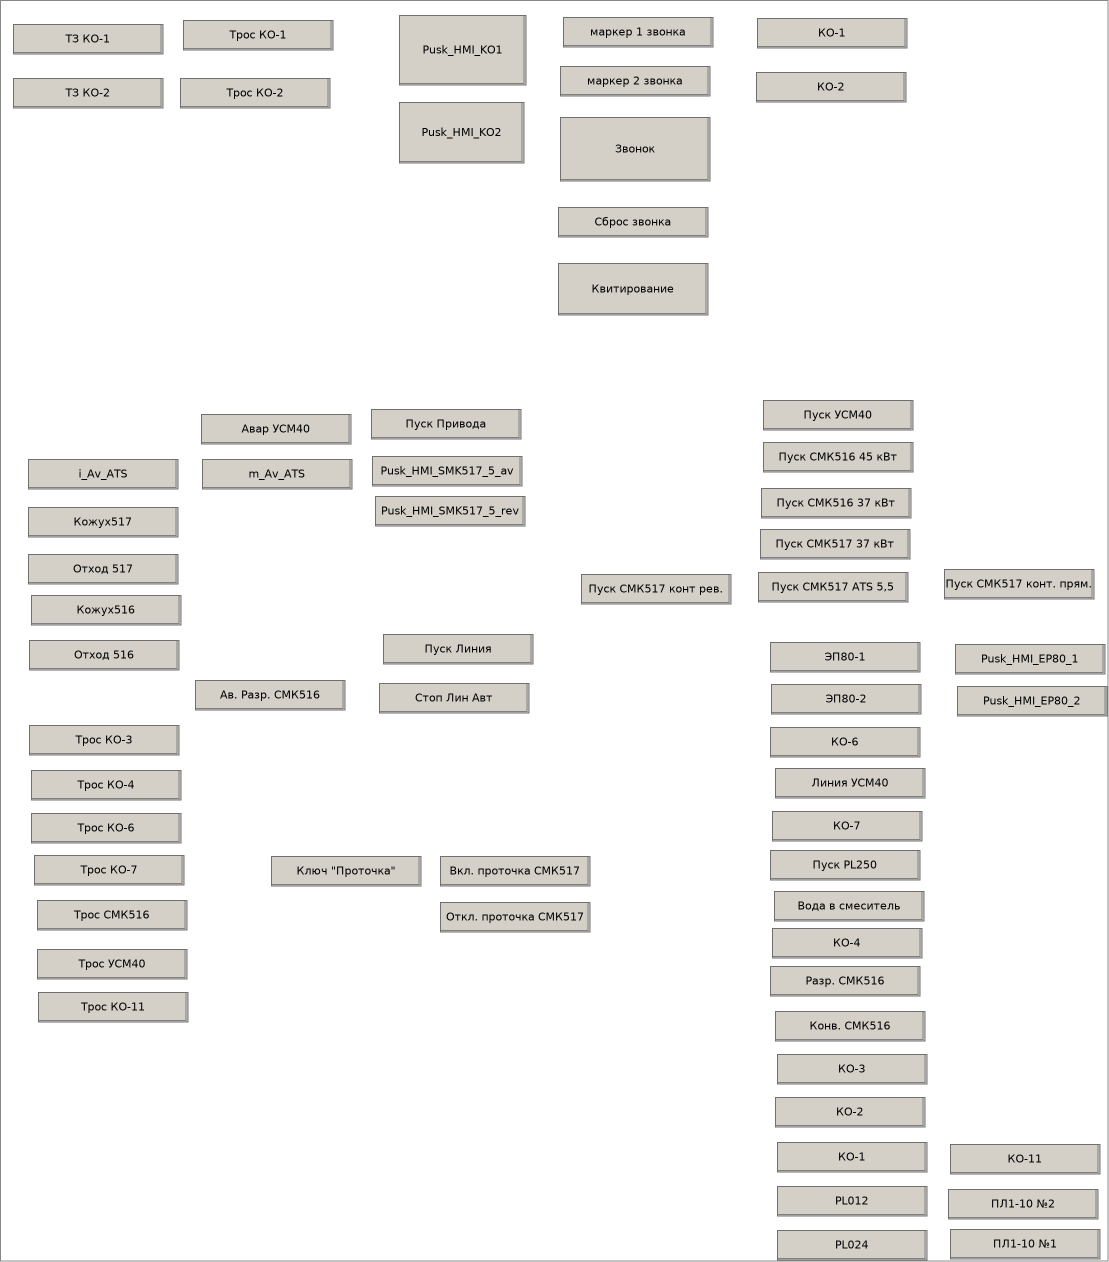
VISUALIZATION VisualizationM  // 1109x1262
    Button (399,15 127x70), "Pusk_HMI_KO1", colour toggle: POU_M.Pusk_HMI_KO1
        toggle POU_M.Pusk_HMI_KO1
    Button (399,102 125x61), "Pusk_HMI_KO2", colour toggle: POU_M.Pusk_HMI_KO2
        toggle POU_M.Pusk_HMI_KO2
    Button (563,17 150x30), "маркер 1 звонка", colour toggle: POU_M.mZV1
    Button (560,66 150x30), "маркер 2 звонка", colour toggle: POU_M.mZV2
    Button (560,117 150x64), "Звонок", colour toggle: IoConfig_Globals_Mapping.q_Zvonok
    Button (757,18 150x30), "КО-1", colour toggle: IoConfig_Globals_Mapping.q_Pusk_KO1
    Button (756,72 150x30), "КО-2", colour toggle: IoConfig_Globals_Mapping.q_Pusk_KO2
    Button (13,24 150x30), "ТЗ КО-1", colour toggle: IoConfig_Globals_Mapping.i_TZ_KO1
        toggle IoConfig_Globals_Mapping.i_TZ_KO1
    Button (13,78 150x30), "ТЗ КО-2", colour toggle: IoConfig_Globals_Mapping.i_TZ_KO2
        toggle IoConfig_Globals_Mapping.i_TZ_KO2
    Button (183,20 150x30), "Трос КО-1", colour toggle: IoConfig_Globals_Mapping.i_Tros_KO1
        toggle IoConfig_Globals_Mapping.i_Tros_KO1
    Button (180,78 150x30), "Трос КО-2", colour toggle: IoConfig_Globals_Mapping.i_Tros_KO2
        toggle IoConfig_Globals_Mapping.i_Tros_KO2
    Button (558,263 150x52), "Квитирование", colour toggle: POU_M.Kvitir_HMI
        toggle POU_M.Kvitir_HMI
    Button (558,207 150x30), "Сброс звонка", colour toggle: POU_M.SbrosZvonka_HMI
        toggle POU_M.SbrosZvonka_HMI
    Button (371,409 150x30), "Пуск Привода", colour toggle: POU_M.Pusk_HMI_Privoda
        toggle POU_M.Pusk_HMI_Privoda
    Button (763,400 150x30), "Пуск УСМ40", colour toggle: IoConfig_Globals_Mapping.q_Pusk_PrivodaUSM40
    Button (770,850 150x30), "Пуск PL250", colour toggle: IoConfig_Globals_Mapping.q_Pusk_PL250
    Button (763,442 150x30), "Пуск СМК516 45 кВт", colour toggle: IoConfig_Globals_Mapping.q_Pusk_SMK516_45
    Button (761,488 150x30), "Пуск СМК516 37 кВт", colour toggle: IoConfig_Globals_Mapping.q_Pusk_SMK516_37
    Button (760,529 150x30), "Пуск СМК517 37 кВт", colour toggle: IoConfig_Globals_Mapping.q_Pusk_SMK517_37
    Button (758,572 150x30), "Пуск СМК517 ATS 5,5", colour toggle: IoConfig_Globals_Mapping.q_Pusk_SMK517_ATS
    Button (774,891 150x30), "Вода в смеситель", colour toggle: IoConfig_Globals_Mapping.q_Vkl_Voda_PL250
    Button (383,634 150x30), "Пуск Линия", colour toggle: POU_M.Pusk_HMI_Liniya
        toggle POU_M.Pusk_HMI_Liniya
    Button (770,642 150x30), "ЭП80-1", colour toggle: IoConfig_Globals_Mapping.q_Pusk_EP80_1
    Button (771,684 150x30), "ЭП80-2", colour toggle: IoConfig_Globals_Mapping.q_Pusk_EP80_2
    Button (772,811 150x30), "КО-7", colour toggle: IoConfig_Globals_Mapping.q_Pusk_KO7
    Button (775,768 150x30), "Линия УСМ40", colour toggle: IoConfig_Globals_Mapping.q_Pusk_LiniyaUSM40
    Button (770,727 150x30), "КО-6", colour toggle: IoConfig_Globals_Mapping.q_Pusk_KO6
    Button (772,928 150x30), "КО-4", colour toggle: IoConfig_Globals_Mapping.q_Pusk_KO4
    Button (770,966 150x30), "Разр. СМК516", colour toggle: POU_M.fbATVRazrSMK516.i_xFwd
    Button (775,1011 150x30), "Конв. СМК516", colour toggle: IoConfig_Globals_Mapping.q_Pusk_KonvSMK516
    Button (777,1054 150x30), "КО-3", colour toggle: IoConfig_Globals_Mapping.q_Pusk_KO3
    Button (775,1097 150x30), "КО-2", colour toggle: IoConfig_Globals_Mapping.q_Pusk_KO2
    Button (777,1142 150x30), "КО-1", colour toggle: IoConfig_Globals_Mapping.q_Pusk_KO1
    Button (777,1186 150x30), "PL012", colour toggle: IoConfig_Globals_Mapping.q_Pusk_PL012
    Button (777,1230 150x30), "PL024", colour toggle: IoConfig_Globals_Mapping.q_Pusk_PL024
    Button (950,1144 150x30), "КО-11", colour toggle: IoConfig_Globals_Mapping.q_Pusk_KO11
    Button (948,1189 150x30), "ПЛ1-10 №2", colour toggle: POU_M.fbATVPL2.i_xFwd
    Button (950,1229 150x30), "ПЛ1-10 №1", colour toggle: POU_M.fbATVPL1.i_xFwd
    Button (955,644 150x30), "Pusk_HMI_EP80_1", colour toggle: POU_M.Pusk_HMI_EP80_1
        toggle POU_M.Pusk_HMI_EP80_1
    Button (957,686 150x30), "Pusk_HMI_EP80_2", colour toggle: POU_M.Pusk_HMI_EP80_2
        toggle POU_M.Pusk_HMI_EP80_2
    Button (372,456 150x30), "Pusk_HMI_SMK517_5_av", colour toggle: POU_M.Pusk_HMI_SMK517_5
        toggle POU_M.Pusk_HMI_SMK517_5
    Button (28,459 150x30), "i_Av_ATS", colour toggle: IoConfig_Globals_Mapping.i_Avar_SMK517_ATS
        toggle IoConfig_Globals_Mapping.i_Avar_SMK517_ATS
    Button (202,459 150x30), "m_Av_ATS", colour toggle: POU_M.m_Avar_SMK517_ATS
    Button (944,569 150x30), "Пуск СМК517 конт. прям.", colour toggle: IoConfig_Globals_Mapping.q_SMK517_Prjamo
    Button (581,574 150x30), "Пуск СМК517 конт рев.", colour toggle: IoConfig_Globals_Mapping.q_SMK517_Revers
    Button (375,496 150x30), "Pusk_HMI_SMK517_5_rev", colour toggle: POU_M.Pusk_HMI_SMK517_5_Rev
        toggle POU_M.Pusk_HMI_SMK517_5_Rev
    Button (28,507 150x30), "Кожух517", colour toggle: IoConfig_Globals_Mapping.i_Kozhuh_SMK517
        toggle IoConfig_Globals_Mapping.i_Kozhuh_SMK517
    Button (31,595 150x30), "Кожух516", colour toggle: IoConfig_Globals_Mapping.i_Kozhuh_SMK516
        toggle IoConfig_Globals_Mapping.i_Kozhuh_SMK516
    Button (195,680 150x30), "Ав. Разр. СМК516", colour toggle: POU_M.fbATVRazrSMK516.q_xAlrm
        toggle POU_M.fbATVRazrSMK516.q_xAlrm
    Button (29,725 150x30), "Трос КО-3", colour toggle: IoConfig_Globals_Mapping.i_Tros_KO3
        toggle IoConfig_Globals_Mapping.i_Tros_KO3
    Button (31,770 150x30), "Трос КО-4", colour toggle: IoConfig_Globals_Mapping.i_Tros_KO4
        toggle IoConfig_Globals_Mapping.i_Tros_KO4
    Button (31,813 150x30), "Трос КО-6", colour toggle: IoConfig_Globals_Mapping.i_Tros_KO6
        toggle IoConfig_Globals_Mapping.i_Tros_KO6
    Button (34,855 150x30), "Трос КО-7", colour toggle: IoConfig_Globals_Mapping.i_Tros_KO7
        toggle IoConfig_Globals_Mapping.i_Tros_KO7
    Button (37,900 150x30), "Трос СМК516", colour toggle: IoConfig_Globals_Mapping.i_Tros_KonvSMK516
        toggle IoConfig_Globals_Mapping.i_Tros_KonvSMK516
    Button (37,949 150x30), "Трос УСМ40", colour toggle: IoConfig_Globals_Mapping.i_TrosLentaUSM40
        toggle IoConfig_Globals_Mapping.i_TrosLentaUSM40
    Button (38,992 150x30), "Трос КО-11", colour toggle: IoConfig_Globals_Mapping.i_Tros_KO11
        toggle IoConfig_Globals_Mapping.i_Tros_KO11
    Button (201,414 150x30), "Авар УСМ40", colour toggle: IoConfig_Globals_Mapping.i_Avar_USM40
        toggle IoConfig_Globals_Mapping.i_Avar_USM40
    Button (271,856 150x30), "Ключ "Проточка"", colour toggle: IoConfig_Globals_Mapping.i_KEY_Protochka
        toggle IoConfig_Globals_Mapping.i_KEY_Protochka
    Button (440,856 150x30), "Вкл. проточка СМК517", colour toggle: IoConfig_Globals_Mapping.i_Vkl_Protoch517
        toggle IoConfig_Globals_Mapping.i_Vkl_Protoch517
    Button (440,902 150x30), "Откл. проточка СМК517", colour toggle: IoConfig_Globals_Mapping.i_Otkl_Protoch517
        toggle IoConfig_Globals_Mapping.i_Otkl_Protoch517
    Button (379,683 150x30), "Стоп Лин Авт", colour toggle: POU_M.StopHMILinAvt
        toggle POU_M.StopHMILinAvt
    Button (28,554 150x30), "Отход 517", colour toggle: IoConfig_Globals_Mapping.i_Othod_SMK517
        toggle IoConfig_Globals_Mapping.i_Othod_SMK517
    Button (29,640 150x30), "Отход 516", colour toggle: IoConfig_Globals_Mapping.i_Othod_SMK516
        toggle IoConfig_Globals_Mapping.i_Othod_SMK516
END_VISUALIZATION
